{attribute 'linkalways'} 
{attribute 'no_explicit_call' := 'This FB is a CLASS and must be accessed using methods or properties'}
{attribute 'enable_dynamic_creation'}
FUNCTION_BLOCK _ETcVnSta EXTENDS EnumDatatypeBase
VAR
	localData : ETcVnSta;
	activeData : REFERENCE TO ETcVnSta;
	enumBaseDatatype : _UDINT(localData);
END_VAR

METHOD PRIVATE AddLocalEnumeration
VAR_INPUT
	Enumeration : T_MAXSTRING;
	Value : ETcVnSta;
END_VAR
AddEnumeration(Enumeration, Value);
END_METHOD

PROPERTY PUBLIC Address : PVOID
GET
Address := ADR(activeData);
END_GET
END_PROPERTY

METHOD PUBLIC ClearReference
VAR_INPUT
END_VAR
activeData REF= localData;
SetBaseDatatypeReference();
END_METHOD

METHOD PUBLIC Clone : I_Datatype
VAR
    pClone : POINTER TO _ETcVnSta;
END_VAR
pClone := __NEW(_ETcVnSta(InitialValue := Value));
Clone := pClone^;
END_METHOD

METHOD FB_init : BOOL
VAR_INPUT
	bInitRetains : BOOL; // if TRUE, the retain variables are initialized (warm start / cold start)
	bInCopyCode : BOOL;  // if TRUE, the instance afterwards gets moved into the copy code (online change)
	InitialValue : ETcVnSta;
END_VAR
localData := InitialValue;
AddBaseDatatype(enumBaseDatatype);
ClearReference();

AddLocalEnumeration('TCVN_STA_CLASSIFIER', ETcVnSta.TCVN_STA_CLASSIFIER);
AddLocalEnumeration('TCVN_STA_NOVELTY_DETECTOR', ETcVnSta.TCVN_STA_NOVELTY_DETECTOR);
AddLocalEnumeration('TCVN_STA_REGRESSOR', ETcVnSta.TCVN_STA_REGRESSOR);
AddLocalEnumeration('TCVN_STA_CLUSTERER', ETcVnSta.TCVN_STA_CLUSTERER);
END_METHOD

PROPERTY PUBLIC Identifier : T_MAXSTRING
GET
Identifier := 'ETcVnSta';
END_GET
END_PROPERTY

METHOD IsEnumeratorValueEqual : BOOL
VAR_INPUT
	Enumerator : I_KeyValueForwardEnumerator;
END_VAR
VAR
	storedValue : ETcVnSta;
END_VAR
IF NOT Enumerator.TryGet(storedValue) THEN
	RETURN;
END_IF

IsEnumeratorValueEqual := storedValue = activeData;
END_METHOD

METHOD PUBLIC MakeReferenceTo
VAR_INPUT
	ReferenceTarget : REFERENCE TO ETcVnSta;
END_VAR
activeData REF= ReferenceTarget;
SetBaseDatatypeReference();
END_METHOD

METHOD PROTECTED SetBaseDatatypeReference
VAR_INPUT
END_VAR
enumBaseDatatype.MakeReferenceTo(activeData);
END_METHOD

PROPERTY PUBLIC Size : UDINT
GET
Size := SIZEOF(activeData);
END_GET
END_PROPERTY

METHOD TryMakeReferenceTo : BOOL
VAR_INPUT
	Target : I_Datatype;
END_VAR
VAR
	targetAsEnum : I_EnumDatatype;
	pTargetData : POINTER TO ETcVnSta;
END_VAR
IF NOT Target.TryResolveAsEnumDatatype(targetAsEnum) THEN
	RETURN;
END_IF

IF targetAsEnum.Identifier <> Identifier THEN
	RETURN;
END_IF

pTargetData := Target.Address;
activeData REF= pTargetData^;
SetBaseDatatypeReference();
TryMakeReferenceTo := TRUE;
END_METHOD

PROPERTY PUBLIC Value : ETcVnSta
GET
Value := activeData;
END_GET
SET
activeData := Value;
END_SET
END_PROPERTY

END_FUNCTION_BLOCK

(* stored: Version 1.1.0.1, ProductVersion 3.1.4024.12
   POU _ETcVnSta: Id {5cdc396d-eeb0-4d4f-a8bb-77662e2d87b9}, SpecialFunc None
   Folder Constructor: Id {e0f832c1-251b-40bd-9482-130b3624ea6b}
   Folder Private: Id {08cfabd9-2000-46e6-8846-ce0431fb1066}
   Folder Protected: Id {43bfb2d8-f0da-43c7-b25d-d56330bb1ca5}
   Method AddLocalEnumeration: Id {66d59224-2c64-4f11-ae5b-49a515a48a99}
   Property Address: Id {070d2a30-3d55-4417-93e3-0ff5505095d0}
   Get Get: Id {70d130f2-1550-4866-939e-8dc44e0a2d34}
   Method ClearReference: Id {de0b2cdf-ffe4-4c40-a918-625d68a742b8}
   Method Clone: Id {9fa42325-ed0d-4c66-9a6a-e6e1d0c371c9}
   Method FB_init: Id {6edadd18-3953-4166-a303-c9c087dde981}
   Property Identifier: Id {d44bbf2a-a3c7-4acc-b019-c46be637d764}
   Get Get: Id {8e80c1bc-ff2d-42e7-bf5a-149096b66c3b}
   Method IsEnumeratorValueEqual: Id {04943906-82d8-4d9c-bda6-ff9ca66cb2df}
   Method MakeReferenceTo: Id {1d0a796a-47f0-4d76-8890-8751badd2c56}
   Method SetBaseDatatypeReference: Id {b30ca750-9525-4be1-a29a-ac4b9e63c8ca}
   Property Size: Id {448e125a-b76d-476c-ae02-27d95af83337}
   Get Get: Id {3355a24c-e67a-4ea1-a6ab-0aed949d73a6}
   Method TryMakeReferenceTo: Id {dded8918-8838-42f2-8866-aee0ebb39d5b}
   Property Value: Id {1abdb52c-92af-4597-9df6-753c71ba6738}
   Get Get: Id {e1c28020-0a9b-4450-b3b7-e34484d58160}
   Set Set: Id {4b46a79d-f209-4740-b67b-d184ed06aac2} *)
